FUNCTION_BLOCK GreenMasterAO EXTENDS GreenMasterAO_Base
VAR_INPUT
END_VAR
VAR_OUTPUT
END_VAR
VAR
	IO_AO_01: AnalogOutput;	
	IO_AO_02: AnalogOutput;	
	IO_AO_03: AnalogOutput;	
	IO_AO_04: AnalogOutput;	
	IO_AO_05: AnalogOutput;	
END_VAR
VAR // added by the converter: edge detectors and wires of the graphical bodies
    _w1, _w2, _w3, _w4, _w5 : INT;
END_VAR


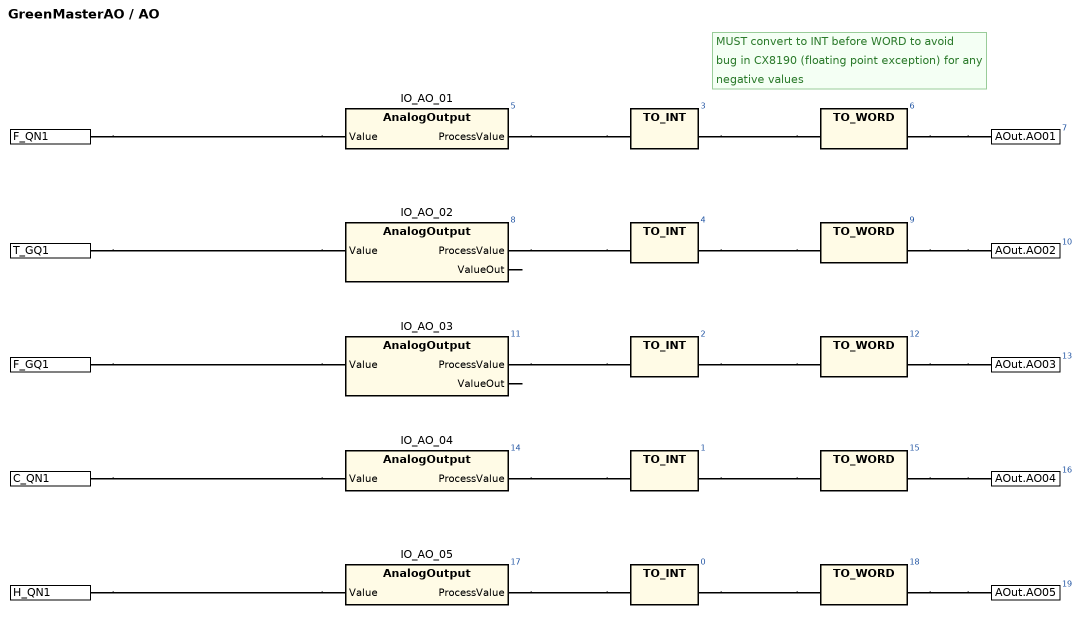
// PAGE AO
_w1 := TO_INT(IO_AO_05.ProcessValue);
_w2 := TO_INT(IO_AO_04.ProcessValue);
_w3 := TO_INT(IO_AO_03.ProcessValue);
// MUST convert to INT before WORD to avoid
// bug in CX8190 (floating point exception) for any
// negative values
_w4 := TO_INT(IO_AO_01.ProcessValue);
_w5 := TO_INT(IO_AO_02.ProcessValue);
IO_AO_01(Value := F_QN1); // AnalogOutput
AOut.AO01 := TO_WORD(_w4);
IO_AO_02(Value := T_GQ1); // AnalogOutput
AOut.AO02 := TO_WORD(_w5);
IO_AO_03(Value := F_GQ1); // AnalogOutput
AOut.AO03 := TO_WORD(_w3);
IO_AO_04(Value := C_QN1); // AnalogOutput
AOut.AO04 := TO_WORD(_w2);
IO_AO_05(Value := H_QN1); // AnalogOutput
AOut.AO05 := TO_WORD(_w1);

METHOD SetOverrideC_QN1 : BOOL
VAR_INPUT
	Override: BOOL;
	OverrideValue: LREAL;
	Parameters: REFERENCE TO GreenMasterBaseParameters;
END_VAR
IO_AO_04.SetOverride2(OverrideIN := Override AND 
	(Parameters.System.Operation.State = SystemStates.Run),
	OverrideValueIN := OverrideValue);
END_METHOD

METHOD SetOverrideF_GQ1 : BOOL
VAR_INPUT
	Override: BOOL;
	OverrideValue: LREAL;
	Parameters: REFERENCE TO GreenMasterBaseParameters;
END_VAR
IO_AO_03.SetOverride2(OverrideIN := Override AND 
	(Parameters.System.Operation.State = SystemStates.Run), OverrideValueIN := OverrideValue);
END_METHOD

METHOD SetOverrideF_QN1 : BOOL
VAR_INPUT
	Override: BOOL;
	OverrideValue: LREAL;
	Parameters: REFERENCE TO GreenMasterBaseParameters;
END_VAR
IO_AO_01.SetOverride2(OverrideIN := Override AND 
	(Parameters.System.Operation.State = SystemStates.Run), OverrideValueIN := OverrideValue);
END_METHOD

METHOD SetOverrideH_QN1 : BOOL
VAR_INPUT
	Override: BOOL;
	OverrideValue: LREAL;
	Parameters: REFERENCE TO GreenMasterBaseParameters;
END_VAR
IO_AO_05.SetOverride2(OverrideIN := Override AND 
	(Parameters.System.Operation.State = SystemStates.Run), OverrideValueIN := OverrideValue);
END_METHOD

METHOD SetOverrideT_GQ1 : BOOL
VAR_INPUT
	Override: BOOL;
	OverrideValue: LREAL;
	Parameters: REFERENCE TO GreenMasterBaseParameters;
END_VAR
IO_AO_02.SetOverride2(OverrideIN := Override AND 
	(Parameters.System.Operation.State = SystemStates.Run), OverrideValueIN := OverrideValue);
END_METHOD

END_FUNCTION_BLOCK

(* stored: Version 1.1.0.1, ProductVersion 3.1.4024.6
   POU GreenMasterAO: Id {ff387c71-d749-4a35-b3f3-c52ada6fced6}, SpecialFunc None
   Method SetOverrideC_QN1: Id {3cd06bd8-e5ee-451d-b3fa-6b642e1750b2}
   Method SetOverrideF_GQ1: Id {9f182b83-0c76-461d-b67a-045d79534555}
   Method SetOverrideF_QN1: Id {f1d64b06-7b8a-4ff2-b775-32e0b65144ba}
   Method SetOverrideH_QN1: Id {3dbe0887-fb81-474e-a5d4-9d6aad747a97}
   Method SetOverrideT_GQ1: Id {a0ebcbe9-0a6e-405e-a5f7-9bc9e521cbc7} *)
